(* PLC project Test, Example PLCOpenEditorExample 1.0, author Laurent Bessard *)
(* stored: companyURL none, productRelease rc1, creationDateTime 2006-09-07T18:52:43, contentDescription Example of PLCOpenEditor usage, version 1, modificationDateTime 2009-09-21T17:43:10, language en-US *)

TYPE MyType : ARRAY[1..16, 1..2] OF INT := [8([-100, 100]), 8([100, -100])];
END_TYPE

TYPE MyType2 : BYTE := 0;
END_TYPE

TYPE MyType3 : (OPEN, CLOSED) := CLOSED;
END_TYPE

TYPE MyType4 : DINT(-4500..4500) := 0;
END_TYPE

TYPE MyType5 : STRUCT
  x : REAL;
  y : REAL;
END_STRUCT;
END_TYPE

FUNCTION_BLOCK FBDTest
  VAR_INPUT
    IN1 : BOOL := false;
    IN2 : BOOL := true;
    IN3 : BOOL;
  END_VAR
  VAR_OUTPUT
    OUT : BOOL;
  END_VAR
  VAR
    SR1 : SR;
  END_VAR
  VAR  (* added by the conversion: wires and edge detectors of the diagram *)
    _AND6_OUT : BOOL;
    _OR8_OUT : BOOL;
    R_TRIG1 : R_TRIG;
  END_VAR

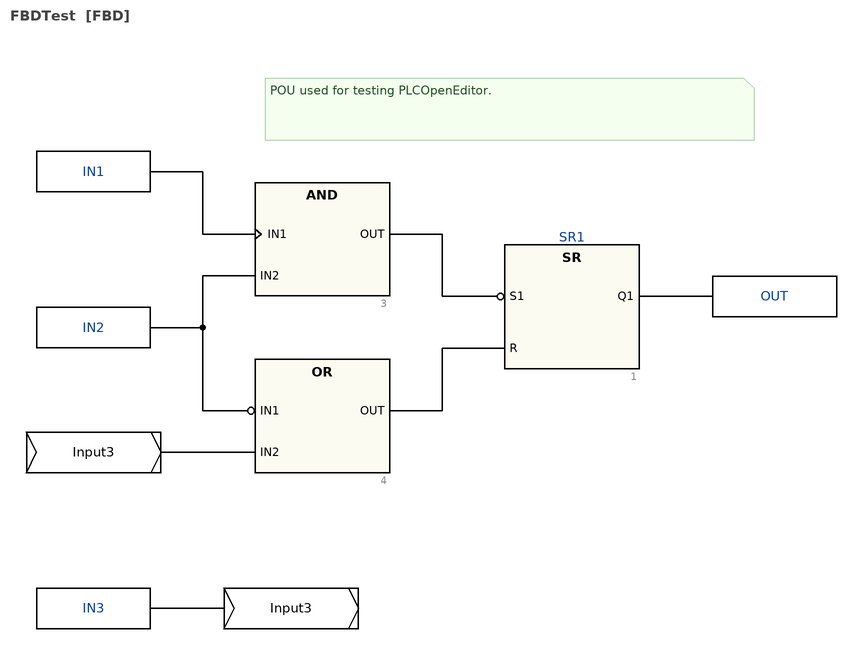
(* FBD diagram, written out as Structured Text *)
(* POU used for testing PLCOpenEditor. *)
SR1(S1 := NOT _AND6_OUT, R := _OR8_OUT);
OUT := SR1.Q1;
R_TRIG1(CLK := IN1);
_AND6_OUT := R_TRIG1.Q AND IN2;
_OR8_OUT := NOT IN2 OR IN3;
END_FUNCTION_BLOCK

FUNCTION LDTest : BOOL
  VAR_INPUT
    IN1 : BOOL;
    IN2 : BOOL;
    IN3 : BOOL;
    IN4 : BOOL;
  END_VAR

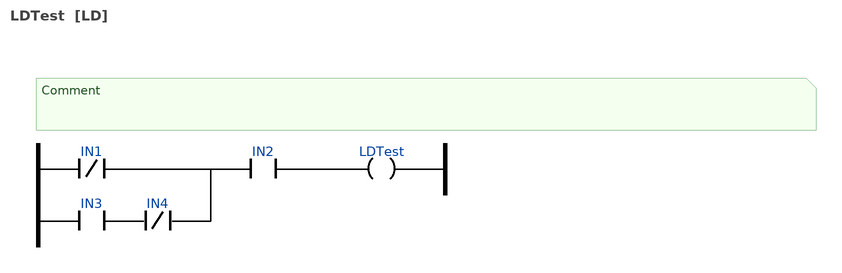
(* LD diagram, written out as Structured Text *)
(* Comment *)
LDTest := (NOT IN1 OR IN3 AND NOT IN4) AND IN2;
END_FUNCTION

FUNCTION ILTest : REAL
  VAR_INPUT
    X1 : REAL;
  END_VAR
  VAR
    Temp : REAL;
  END_VAR
  VAR_INPUT
    X2 : REAL;
    Y1 : REAL;
    Y2 : REAL;
    TMax : REAL;
  END_VAR
  VAR_OUTPUT
    ERROR : BOOL;
  END_VAR

     LD   Y1
     SUB  Y2     (* Substract Y2 from Y1 *)
     ST   Temp   (* Store Y1-Y2 in Temp *)
     MUL  Temp   (* Multiply by Temp to square *)
     ADD( X1     (* Defer ADD *)
     SUB  X2     (* Substract X1 from X2 *)
     ST   Temp   (* Store X1-X2 in Temp *)
     MUL  Temp   (* Multiply by Temp to square *)
     )
     SQRT        (* Call Square root fun *)
     ST   ILTest (* Setup function result *)
     GT   TMax   (* Greater than TMax ? *)
     JMPC ERR    (* Yes, Jump to Error *)
     S    ERROR  (* Set ERROR *)
     RET         (* Normal return *)
ERR: RET         (* Error return, ENO not set *)

          
END_FUNCTION

PROGRAM SFCTest
  VAR
    IN1 : BOOL;
  END_VAR
  VAR_INPUT
    IN2 : BOOL;
    IN3 : BOOL;
    IN4 : BOOL;
    IN5 : BOOL;
  END_VAR
  VAR
    SR1 : SR;
  END_VAR
  VAR  (* added by the conversion: wires and edge detectors of the diagram *)
    R_TRIG1 : R_TRIG;
  END_VAR

(* transition TR2 *)
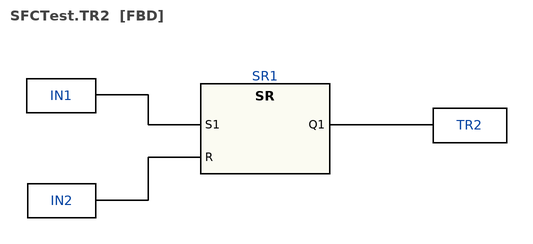
(* FBD diagram, written out as Structured Text *)
SR1(S1 := IN1, R := IN2);
TR2 := SR1.Q1;
(* transition TR3 *)
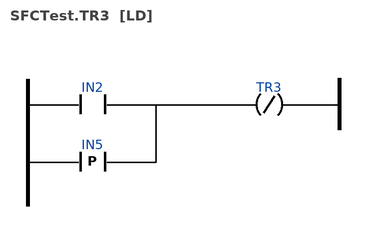
(* LD diagram, written out as Structured Text *)
R_TRIG1(CLK := IN5);
TR3 := NOT (IN2 OR R_TRIG1.Q);
(* transition TR4 *)
    LD  IN3
    AND IN4

              
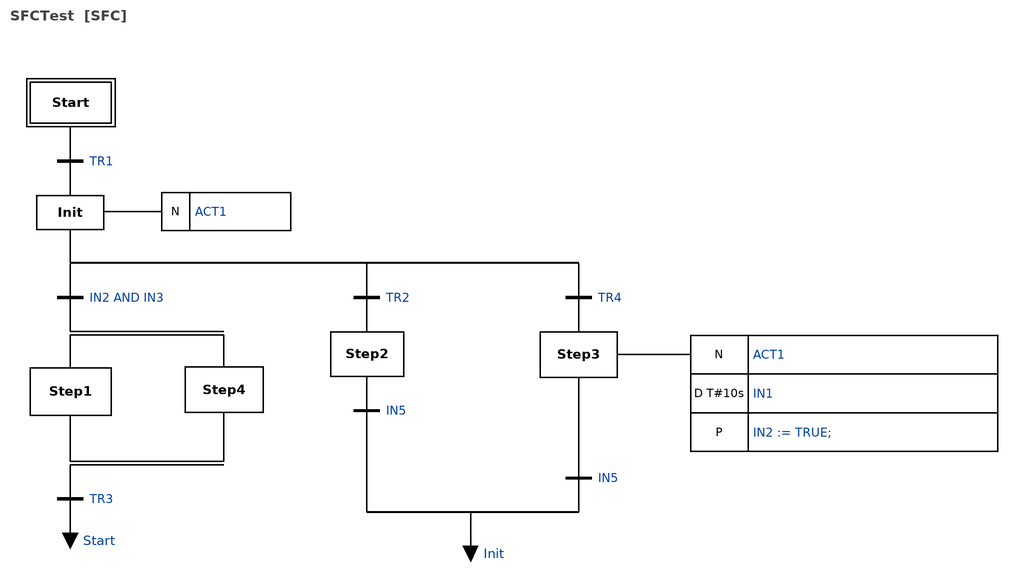
INITIAL_STEP Start:
END_STEP
TRANSITION FROM Start TO Init  (* TR1 *)
  := AND(IN1, IN2, IN3);
END_TRANSITION
STEP Init:
  ACT1(N);
END_STEP
TRANSITION FROM Init TO (Step1, Step4)
  := IN2 AND IN3;
END_TRANSITION
TRANSITION (PRIORITY := 1) FROM Init TO Step2
  := TR2;
END_TRANSITION
TRANSITION FROM Init TO Step3
  := TR4;
END_TRANSITION
STEP Step2:
END_STEP
TRANSITION FROM Step2 TO Init
  := IN5;
END_TRANSITION
STEP Step3:
  ACT1(N, IN5);
  IN1(D, T#10s);
  STEP3_INLINE1(P);
END_STEP
ACTION STEP3_INLINE1:
  IN2 := TRUE;
END_ACTION
TRANSITION FROM Step3 TO Init
  := IN5;
END_TRANSITION
STEP Step4:
END_STEP
STEP Step1:
END_STEP
TRANSITION FROM (Step1, Step4) TO Start
  := TR3;
END_TRANSITION

ACTION ACT1:
IF IN1 THEN
  IN2 := 1;
ELSE
  IN3 := 1;
END_IF;

              
END_ACTION
END_PROGRAM

FUNCTION_BLOCK STTest
  VAR_INPUT
    Collision : BOOL;
    Gate : BOOL;
    Pump : BOOL;
    Temp : REAL;
  END_VAR
  VAR_OUTPUT
    Speed : INT;
    PumpSpeed : INT;
    Brakes : BOOL;
    Control_State : BOOL;
  END_VAR

IF Collision THEN
  Speed := 0;
  Brakes := TRUE;
END_IF;

IF (Gate = open) AND
    (Pump = TRUE) AND (Temp > 200.0) THEN
  Control_State := TRUE;
ELSE
  Control_State := FALSE;

  PumpSpeed := 10.0;
END_IF;

          
END_FUNCTION_BLOCK

CONFIGURATION ConfigTest
  VAR_GLOBAL
    Toto AT %MW10 : INT;
    Tutu AT %MX20 : BOOL;
  END_VAR
  RESOURCE ResourceTest ON PLC
    VAR_GLOBAL
      Titi AT %MW30 : INT;
    END_VAR
    TASK Toto(SINGLE := Tutu, PRIORITY := 6);
    PROGRAM Program1 WITH Toto : SFCTest;
  END_RESOURCE
END_CONFIGURATION
